// TIA Portal V17 export
// export: Created 2023-04-11T09:33:31.7415111Z, ExportSetting WithDefaults, DisplayName Totally Integrated Automation Portal, DisplayVersion V17 Update 3, DisplayName TIA Portal Openness, DisplayVersion V17 Update 3, DisplayName TIA Portal Version Control Interface, DisplayVersion V17, DisplayName SINAMICS Startdrive Advanced, DisplayVersion V17 Update2, DisplayName SINAMICS Startdrive G130, G150, S120, S150, SINAMICS MV, S210, DisplayVersion V17 Update2, DisplayName SINAMICS Startdrive G110M, G120, G120C, G120D, G120P, G115D, DisplayVersion V17 Update2, DisplayName STEP 7 Professional, DisplayVersion V17 Update 3, DisplayName STEP 7 Safety, DisplayVersion V17, DisplayName WinCC UA Professional, DisplayVersion V17 Update 3
FUNCTION "FC_rst8" : Void   // FC23, LAD
{ S7_Optimized_Access := 'TRUE' }
VERSION : 0.1
// stored: AutoNumber true, IsIECCheckEnabled false, SetENOAutomatically false, UDAEnableTagReadback false
   VAR_OUTPUT
      rst0 : Bool;
      rst1 : Bool;
      rst2 : Bool;
      rst4 : Bool;
      rst5 : Bool;
      rst6 : Bool;
      rst7 : Bool;
      rst8 : Bool;
   END_VAR
BEGIN

REGION Network 1
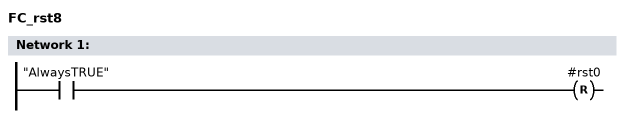
   RUNG wire#powerrail
      Contact( "AlwaysTRUE" )
      R_Coil( #rst0 )
   END_RUNG
   // the same network as SCL:
   IF "AlwaysTRUE" THEN #rst0 := FALSE; END_IF;
END_REGION
END_FUNCTION
